Yaskawa INFORM job: TC_COLDSTART.JBI

/JOB
//NAME TC_COLDSTART
//POS
///NPOS 0,0,0,0,0,0
//INST
///DATE 2026/02/10 15:13
///ATTR SC,RW
///GROUP1 RB1
NOP
'WAIT FAULT OFF
WAIT IN#(207)=OFF
TIMER T=0.10
'WAIT MOTOR ENABLED
WAIT IN#(206)=ON
TIMER T=0.20
'SET NULL TOOL
DOUT OG#(26) 0
TIMER T=0.10
'FLUSH OUTPUT COMMANDS
DOUT OG#(27) 0
TIMER T=0.10
'SET HOME COMMAND
DOUT OG#(27) 2
TIMER T=0.10
'RESET HOME COMMAND
DOUT OG#(27) 0
'WAIT FOR HOME
WAIT IN#(205)=ON
TIMER T=0.10
'WAIT FOR IDLE STATE
WAIT IN#(209)=OFF
WAIT IN#(210)=ON
WAIT IN#(211)=OFF
TIMER T=0.20
END
